{attribute 'enable_dynamic_creation'}
FUNCTION_BLOCK FB_Circle IMPLEMENTS I_Shape
VAR_INPUT
END_VAR
VAR_OUTPUT
END_VAR
VAR
END_VAR

METHOD M_Draw : BOOL
ADSLOGSTR(ADSLOG_MSGTYPE_HINT, 'Draw circle', '');
M_Draw := TRUE;
END_METHOD

END_FUNCTION_BLOCK

(* stored: Version 1.1.0.1, ProductVersion 3.1.4024.12
   POU FB_Circle: Id {2630a463-c142-4a6a-81ee-b7dcaa9a3c1d}, SpecialFunc None
   Method M_Draw: Id {5874aed3-bb9c-4bb3-9b3f-d577d5929cd2} *)
